RoboDK station: kr30 cnc 070119 halp.rdk

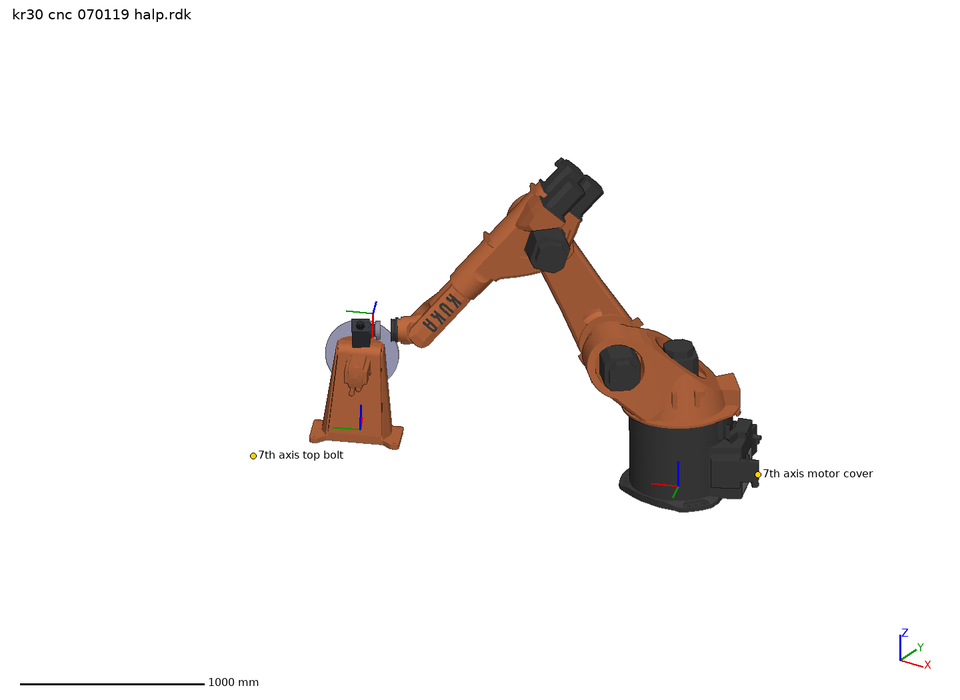
[picture v0: the station drawn from its stored meshes, robots at their saved joint values, targets as dots, program paths as lines]
Station kr30 cnc 070119 halp. Poses are relative to the parent item; angles as X-Y-Z fixed-axis rotations.
  - frame KUKA KR 30 HA Base at (1535.48, 628.29, -1072.61) mm, rotated rx 0 ry 0 rz -156.31 deg
    - robot KUKA KR 30 HA: 6 axes, payload 30 kg, reach 2033 mm, repeatability 0.05 mm, weight 665 kg
        modified DH rows (alpha deg, a mm, theta deg, d mm): 0, 0, 0, 815; -90, 350, 0, 0; 0, 850, -90, 0; -90, 145, 0, 820; 90, 0, 0, 0; -90, 0, 180, 170
        joint limits [-185, -135, -120, -350, -119, -350] to [185, 35, 158, 350, 119, 350]; home [0, -90, 90, 0, 0, 0]; saved at [-21.51, -62.12, 108.88, 165.58, 46.68, -127.57]
      - tool 1/2" End Mill TCP, TCP at (337.71, -2.2, 160.57) mm, rotated rx 0 ry 90 rz 0 deg, size 415.8 x 102 x 153.6 mm
    - target 7th axis top bolt (joint target) at (1966.13, 1947.63, 927.26) mm, rotated rx -179.2 ry 6.72 rz -171.11 deg; joints [-17.018, -71.525, 110.046, 168.711, 45.865, -170.331, 883.939] of KUKA KR 30 HA
    - target 7th axis motor cover (joint target) at (-417, -111.35, 57.2) mm, rotated rx -135.46 ry -1.69 rz -48.75 deg; joints [-33.388, -54.543, 96.086, 147.711, 45.276, -113.831, 883.939] of KUKA KR 30 HA
  - frame KUKA KP1 MD250 Base at (172.34, -439.05, -684.5) mm, rotated rx 2 ry 0.52 rz 120.23 deg
    - robot KUKA KP1 MD250: 1 axes, payload 250 kg
        modified DH rows (alpha deg, a mm, theta deg, d mm): 0, 0, 0, 0
        base shift (70, 10, 428) mm, rotated rx 0 ry 90 rz -2 deg
        joint limits [-3600] to [3600]; home [0]; saved at [-3600]
      - frame Frame 2 at (0, 0, 500) mm
  - machining project Machining Settings: C:/Users/liqui/Downloads/070119 rotary tower 01.apt | rotZ(0) | rotX(0)*rotY(0) | rotz(0)
